// TIA Portal V16 export
// export: Created 2022-09-01T14:27:02.4834896Z, ExportSetting WithDefaults, DisplayName Totally Integrated Automation Portal, DisplayVersion V16, DisplayName TIA Portal Version Control Interface, DisplayVersion V16, DisplayName TIA Portal Openness, DisplayVersion V16, DisplayName STEP 7 Professional, DisplayVersion V16, DisplayName STEP 7 Safety, DisplayVersion V16, DisplayName WinCC Advanced, DisplayVersion V16
DATA_BLOCK "Dados_Bombas"   // DB11
{ S7_Optimized_Access := 'TRUE' }
VERSION : 0.1
// stored: AutoNumber true, IsOnlyStoredInLoadMemory false, IsRetainMemResEnabled false, IsWriteProtectedInAS false, MemoryReserve 100
   VAR
      CONV_T_ALTERNANCIA_BOMBAS : Time;
      HORAS_TON_B2 : Int;
      HORAS_TON_B3 : Int;
      HORAS_TON_B1 : Int;
   END_VAR
BEGIN
END_DATA_BLOCK
